PROGRAM PDMctr
VAR
	FB_PDMSCtr:FB_PDMSCtr;

	TonWrite: TON;
	TonWriteQ: BOOL;

END_VAR

FB_PDMSCtr(
	stLightCtr:= stLightCtr, 
	strNetID:=stSystem.strNetID , 
	uiSlaveAddr:=1010, 
	wIndex:= 16#8000, 
	wstrCommPara=> );

END_PROGRAM

(* stored: Version 1.1.0.1, ProductVersion 3.1.4024.12
   POU PDMctr: Id {5d420222-756d-4c5d-b75c-0781e256448e}, SpecialFunc None *)
